FUNCTION_BLOCK EL3403
VAR
	_io : EL3403_Data;
	{attribute addProperty Name "WcState"}
	_wcState : WcStateInputToggle;
	{attribute addProperty Name "Info data"}
	_infoData : InfoDataAds;
END_VAR

PROPERTY IO : REFERENCE TO EL3403_Data
GET
IO REF= _io;
END_GET
END_PROPERTY

PROPERTY WcState : REFERENCE TO WcStateInputToggle
GET
WcState REF= _wcState;
END_GET
END_PROPERTY

END_FUNCTION_BLOCK

(* stored: Version 1.1.0.1, ProductVersion 3.1.4024.9
   POU EL3403: Id {08cc460e-2a4c-0450-194f-ccb7a2032697}, SpecialFunc None
   Property IO: Id {afe5a081-534c-0283-2ef6-c7dc86a4f257}
   Get Get: Id {28e2eb41-063d-0ad4-3151-2f9b6154af84}
   Property WcState: Id {3c64c7dc-a13e-0f44-0341-8aee230d0f1d}
   Get Get: Id {57615cb1-c2f2-0ea9-1d94-40e662641d2a} *)
